// TIA Portal V20 export
DATA_BLOCK "IDB_FB_Merging"   // DB39
// stored: InstanceOfName LineC1.FB_Merging, InstanceOfType FB, Namespace LineC1
"LineC1.FB_Merging"
   // VAR
   //    Merge : "Global.FB_Merging";
   // END_VAR
BEGIN
END_DATA_BLOCK
